// TIA Portal V20 export
TYPE "LER_typeStatusEm5"
// stored: Access Published
   STRUCT
      cathodePnP1XCamEnabled : Bool;
      cathodePnP1ZCamEnabled : Bool;
      cathodePnP2XCamEnabled : Bool;
      cathodePnP2ZCamEnabled : Bool;
      cathodeDownComplete1 : Bool;
      cathodeDownComplete2 : Bool;
      cathodeSupplyCheck : Bool;
      cathodeFinishCheck : Bool;
      cathodeSupplyComplete : Bool;
      cathodeFinishComplete : Bool;
      cathodeReady : Bool;
      cathodeRequest : Bool;
      stackJobCompleteChecked : Bool;
      stopRequest : Bool;
      stopComplete : Bool;
      cathodePnP1HomePos : Bool;
      cathodePnP1WorkPos : Bool;
      cathodePnP2HomePos : Bool;
      cathodePnP2WorkPos : Bool;
      cathodeAvoidPos : Bool;
      cathodeReelcutRequest : Bool;
      cathodeStartCase : DInt;
      cathodePnPXStart : LReal := 0.0;
      cathodePnPXEnd : LReal := 75.0;
      cathodePnPZDownStart : LReal := 65.0;
      cathodePnPZDownEnd : LReal := 75.0;
      cathodePnPZUpStart : LReal := 90.0;
      cathodePnPZUpEnd : LReal := 100.0;
      cathodePnP1ZOnPos : LReal := 5.0;
      cathodePnP1ZOffPos : LReal := 5.0;
      cathodeReelCutOnPos : LReal := 5.0;
      cathodePnP2ZOnPos : LReal := 5.0;
      cathodePnP2ZOffPos : LReal := 5.0;
      cathodeAlignOnPos : LReal := 5.0;
      cathodeAlignOffPos : LReal := 5.0;
      cathodeVisionTrigger : LReal := 5.0;
      cathodeVisionClean : LReal := 5.0;
   END_STRUCT;
END_TYPE
